// TIA Portal V16 export
// export: Created 2022-11-17T11:56:29.5480859Z, ExportSetting WithDefaults, DisplayName Totally Integrated Automation Portal, DisplayVersion V16 Update 6, DisplayName TIA Portal Version Control Interface, DisplayVersion V16 Update 2, DisplayName TIA Portal Openness, DisplayVersion V16 Update 6, DisplayName SINAMICS Startdrive Advanced, DisplayVersion V16 Update 5, DisplayName SINAMICS Startdrive G130, G150, S120, S150, SINAMICS MV, S210, DisplayVersion V16 Update 5, DisplayName SINAMICS Startdrive G110M, G120, G120C, G120D, G120P, G115D, DisplayVersion V16 Update 5, DisplayName STEP 7 Professional, DisplayVersion V16 Update 6, DisplayName STEP 7 Safety, DisplayVersion V16, DisplayName WinCC Advanced, DisplayVersion V16 Update 6
FUNCTION "Centrador_Paletes" : Void   // FC17, LAD
{ S7_Optimized_Access := 'TRUE' }
VERSION : 0.1
// stored: AutoNumber true, IsIECCheckEnabled false, SetENOAutomatically false, UDAEnableTagReadback false
   VAR_TEMP
      Detetor_Palete : Bool;
      Comando_Tapete_Centrador : Bool;
      Start : Bool;
      Setpoint : Real;
      ActVelocity : Real;
      RefSpeed : Real;
   END_VAR
   VAR_TEMP   // added for the SCL form of the ladder/FBD networks
      _w1 : Bool;
   END_VAR
BEGIN

REGION Network 1: Motor tapete de rolos do centrador
   // Tapete só anda se ambas as barras centradoras estiverem na posição aberta e pára quando deteta palete
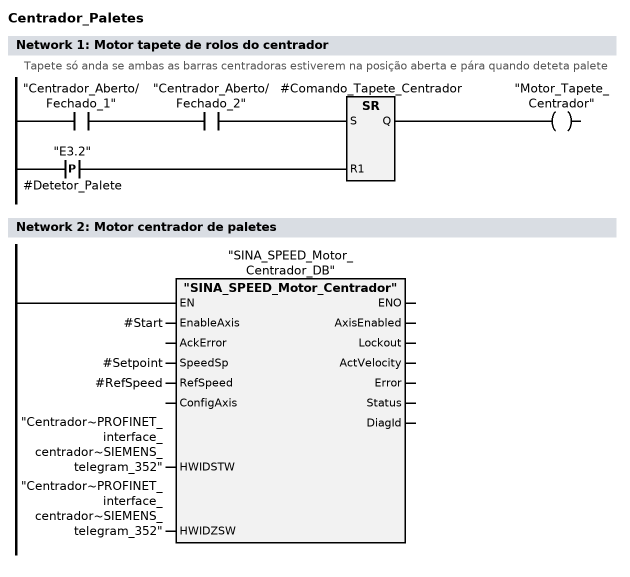
   RUNG wire#powerrail
      Contact( "Centrador_Aberto/Fechado_1" )
      Contact( "Centrador_Aberto/Fechado_2" )
      S_SR(operand := #Comando_Tapete_Centrador, r1 := wire#w1)
      Coil( "Motor_Tapete_Centrador" )
   END_RUNG
   RUNG wire#powerrail
      P_Contact(operand := "E3.2", bit := #Detetor_Palete)
   END_RUNG wire#w1
   // the same network as SCL:
   #_w1 := "E3.2" AND NOT #Detetor_Palete;   // rising edge of "E3.2"
   #Detetor_Palete := "E3.2";
   IF "Centrador_Aberto/Fechado_1" AND "Centrador_Aberto/Fechado_2" THEN
       #Comando_Tapete_Centrador := TRUE;   // SR flip-flop
   END_IF;
   IF #_w1 THEN #Comando_Tapete_Centrador := FALSE; END_IF;
   "Motor_Tapete_Centrador" := #Comando_Tapete_Centrador;
END_REGION

REGION Network 2: Motor centrador de paletes
   RUNG wire#powerrail
      "SINA_SPEED_Motor_Centrador_DB"(EnableAxis := #Start, AckError :=, SpeedSp := #Setpoint, RefSpeed := #RefSpeed, ConfigAxis :=, HWIDSTW := "Centrador~PROFINET_interface_centrador~SIEMENS_telegram_352", HWIDZSW := "Centrador~PROFINET_interface_centrador~SIEMENS_telegram_352", AxisEnabled =>, Lockout =>, ActVelocity =>, Error =>, Status =>, DiagId =>)
   END_RUNG
   // the same network as SCL:
   "SINA_SPEED_Motor_Centrador_DB"(EnableAxis := #Start,   // "SINA_SPEED_Motor_Centrador"
                           SpeedSp := #Setpoint,
                           RefSpeed := #RefSpeed,
                           HWIDSTW := "Centrador~PROFINET_interface_centrador~SIEMENS_telegram_352",
                           HWIDZSW := "Centrador~PROFINET_interface_centrador~SIEMENS_telegram_352");
END_REGION
END_FUNCTION
